// TIA Portal V19 export
TYPE "Prod_Item_small"
// stored: Access Published
   STRUCT
      O_ID : DInt;   // ID PLC per riferimento allìordine di produzione
      PPrf_No : DInt;   // Numero del programma profillo che corrisponde al codice MES del prodotto da eseguire
      MES_IDP : String[30];   // ID MES per riferimento all'ordine di prosuzione
      MES_PPrf_Name : String[20];   // Nome dell programma profilo richiesto da MES (es.C040x45x1.25)
      Beam_Code : Int;   // Codice Pezzo: 0= SG formato da una singola parte; 1= C/S = Formato da due parti accoppiate
      Beams_W_A : Real;   // Dim. base pezzo (W) = Altezza in impilamento (A)
      Beams_H_B : Real;   // Dim. altezza pezzo (H) = base in impilamento (B)
      Beams_Thickness : Real;   // Spessore lamiera del profilo
      Beams_Len_Min : Real;   // Lunghezza pezzo - Tolleranza minima
      Beams_Len_Max : Real;   // Lunghezza pezzo + Tolleranza massima
      Beams_Len : Real;   // Lunghezza pezzi richiesta
      Parts_Len : Real;   // Lunghezza delle parti con target al centro della tolleranza richiesta
      Parts_Tol : Real;   // Tolleranza su lunghezza parte tagliata
      PackLayout_BeamsPerLayer : Int;   // Schema del pacco - Numero pezzi per strato
      PackLayout_Layers_Qty : Int;   // Schema del pacco - Numero strati
   END_STRUCT;
END_TYPE
